SUBAPPLICATION Uebung_003a_sub (* IX auf QX (generisch) *)
  (* Standard: 61499-2 *)
  (* Version 1.0, 2023-10-23, franz *)
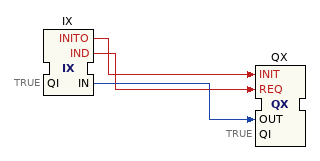
  FBS
    QX : QX(QI := TRUE);
    IX : IX(QI := TRUE);
  END_FBS
  EVENT_CONNECTIONS
    IX.INITO TO QX.INIT;
    IX.IND TO QX.REQ;
  END_CONNECTIONS
  DATA_CONNECTIONS
    IX.IN TO QX.OUT;
  END_CONNECTIONS
END_SUBAPPLICATION
